// TIA Portal V20 export
// export: Created 2026-07-10T11:12:34.7291477Z, ExportSetting WithDefaults, DisplayName Totally Integrated Automation Portal, DisplayVersion V20, DisplayName TIA Portal Openness, DisplayVersion V20, DisplayName TIA Portal Version Control Interface, DisplayVersion V20, DisplayName STEP 7 Professional, DisplayVersion V20, DisplayName STEP 7 Safety, DisplayVersion V20, DisplayName WinCC Basic/Comfort/Advanced, DisplayVersion V20, DisplayName WinCC Unified, DisplayVersion V20
FUNCTION_BLOCK "ChlorMode"   // FB5, SCL
{ S7_Optimized_Access := 'TRUE' }
VERSION : 0.1
// stored: AutoNumber true, IsIECCheckEnabled false, IsRetainMemResEnabled false, MemoryReserve 100, SetENOAutomatically false, UDAEnableTagReadback false
   VAR
      WaterLevel : Real;
      WaterPulse_RT { S7_SetPoint := 'True'} : R_TRIG;
      PulseSetpoint { S7_SetPoint := 'True'} : Real;
      FreqTON { S7_SetPoint := 'True'} : TON_TIME;
      LevelAlarm { S7_SetPoint := 'True'} : Bool;
      DelayTOF { S7_SetPoint := 'True'} : TOF_TIME;
      PulseGen { S7_SetPoint := 'True'} : TP_TIME;
      DoserValue { S7_SetPoint := 'True'} : Real := 0.0;
      DoserPreValue : Real;
      StopTrig { S7_SetPoint := 'True'} : R_TRIG;
      StartTrig { S7_SetPoint := 'True'} : R_TRIG;
      ChlorMeasurment { S7_SetPoint := 'True'} : "ChlorMeasurment";
      BlockDosing { S7_SetPoint := 'True'} : Bool;
      EnableMeasureTime : Real;
      BlockDosingTime : Real;
   END_VAR
   VAR CONSTANT
      Freq : UDInt := 10;
   END_VAR
BEGIN
   "DoserOut" := FALSE;

   //#WaterPulse_RT(CLK := "WaterCounterOutPulse");
   #ChlorMeasurment(blockDosing=>#BlockDosing);

   "Config".DiOxydeDosing := REAL_TO_DWORD("MB".Table.ChlorationParams.ActualDose);
   "Config".DiOxydeDosing := ROL(IN := "Config".DiOxydeDosing, N := 16);
   "ModbusMaster"(REQ := "ModbusLoad".DONE,
                  MB_ADDR := 1,
                  MODE := 1,
                  DATA_ADDR := 40055,
                  DATA_LEN := 2,
                  DATA_PTR := "Config".DiOxydeDosing);

   IF NOT "MB".Table.HMI_ChlorModeOn OR NOT "MB".Table.Chlor_AutoMode THEN
       "MB".Table.ChlorationParams.ActualDose := 0;

   END_IF;

   IF "MB".Table.HMI_Chlor_ChooseTank = 0 THEN
       #LevelAlarm := "MB".Table.Alarms_RCV1Min OR "MB".Table.Alarms_RCV1Max;
   END_IF;

   IF "MB".Table.HMI_Chlor_ChooseTank = 1 THEN
       #LevelAlarm := "MB".Table.Alarms_RCV2Min OR "MB".Table.Alarms_RCV2Max;
   END_IF;

   "MB".Table.DoserNotWork := (
       #LevelAlarm OR
       "MB".Table.Alarms_ChlorLargeConsumption OR
       #BlockDosing OR
       "MB".Table.CriticalMeasureON
       );

   REGION ChlorationAlgorithm
       // Statement section REGION
       #StartTrig(CLK := "MB".Table.Chlor_StartManual);
       IF #StartTrig.Q THEN
           #DoserValue := 0;
           #DoserPreValue := "MB".Table.Doser1_DailyValue;
       END_IF;

       IF "MB".Table.Chlor_AutoMode THEN
           #FreqTON(IN := #PulseSetpoint > 0,
                    PT := UDINT_TO_DINT(500));
           IF "MB".Table.HMI_ChlorModeOn THEN
               IF "Config".WaterPulseDuble THEN
                   "Config".WaterPulseDuble := FALSE;
                   #PulseSetpoint += "MB".Table.ChlorationParams.ActualDose / "MB".Table.Chlor_PulseWeight_1 * "MB".Table.WaterCounterOut_PulseValue;
               END_IF;



           END_IF;
           IF #FreqTON.Q THEN
               IF #PulseSetpoint >= 0 THEN
                   #PulseGen(IN := #FreqTON.Q,
                             PT := UDINT_TO_DINT(250));
                   #PulseSetpoint -= 1;
               END_IF;
               RESET_TIMER(#FreqTON);
           END_IF;

           IF #PulseGen.Q THEN
               "DoserOut" := True;
               RESET_TIMER(#PulseGen);
           END_IF;
       ELSIF NOT "MB".Table.Chlor_AutoMode AND "MB".Table.Chlor_StartManual THEN
           #StopTrig(CLK := #DoserValue > "MB".Table.Chlor_ManualSetpoint_1 * 1000);
           IF #StopTrig.Q THEN
               "MB".Table.HMI_WeightAlarmReset := 1;
               "MB".Table.Chlor_StartManual := 0;
               RETURN;
           END_IF;

           #DoserValue := "MB".Table.Doser1_DailyValue - #DoserPreValue;
           #FreqTON(IN := #DoserValue < "MB".Table.Chlor_ManualSetpoint_1 * 1000,
                    PT := UDINT_TO_DINT(500));
           IF #FreqTON.Q THEN
               #PulseGen(IN := #FreqTON.Q,
                         PT := UDINT_TO_DINT(250));
               RESET_TIMER(#FreqTON);
           END_IF;

           IF #PulseGen.Q THEN
               IF #DoserValue < "MB".Table.Chlor_ManualSetpoint_1 * 1000 THEN
                   "DoserOut" := True;
                   RESET_TIMER(#PulseGen);
               END_IF;
           END_IF;
       END_IF;
   END_REGION



   IF "MB".Table.DoserNotWork AND "MB".Table.Chlor_AutoMode THEN
       #PulseSetpoint := 0;
       "MB".Table.ChlorationParams.ActualDose := 0;
   END_IF;
END_FUNCTION_BLOCK
